FUNCTION ScaleAndRound : REAL
VAR_INPUT
    realValue 	: REAL;              // Die zu rundende REAL-Zahl
    scaleFactor : INT;           // Rundungsfaktor
END_VAR

ScaleAndRound := INT_TO_REAL(REAL_TO_INT(realValue * scaleFactor)) / scaleFactor;

END_FUNCTION

(* stored: Version 1.1.0.1
   POU ScaleAndRound: Id {5b993068-a871-4d85-b067-4291ff7e8272}, SpecialFunc None *)
